{attribute 'GeneratedUsingTerminal: IODEVICETYPE_ETHERCATPROT'}
{attribute addProperty BoxType "IODEVICETYPE_ETHERCATPROT"}
{attribute addProperty Id "Term_26_EK1100Term_26_EK1100_99E5D94A13Box_29_EP1008_0001EP1008_78E8D3DD12Box_30_EP1008_0001EP1008_78E8D3DD12Box_31_EP1008_0001EP1008_78E8D3DD12Box_32_EP1008_0001EP1008_78E8D3DD12Box_33_EP1008_0001EP1008_78E8D3DD12Box_34_EP1008_0001EP1008_78E8D3DD12Box_35_EP1008_0001EP1008_78E8D3DD12Box_36_EP1008_0001EP1008_78E8D3DD12Box_37_EP1008_0001EP1008_78E8D3DD12Box_38_EP1008_0001EP1008_78E8D3DD12SyncUnitsSyncUnits_1397309536InputsInputs_A65FACA410OutputsOutputs_23C0ED1D6InfoDataInfoData_84133AC922"}
{attribute addProperty CRC "3568369493"}
{attribute addProperty Size "207"}
{attribute addProperty Name "Device 2 (EtherCAT)"}
TYPE Device_2_EtherCAT_D4B0FF55 EXTENDS TcoIo.EtcMasterBase_62654B43 :
STRUCT
	{attribute addProperty Name "Term 26 (EK1100)"}
	{attribute addProperty PreviousPort "Device 2 (EtherCAT) : Master"}
	Term_26_EK1100 : Term_26_EK1100_99E5D94A;
	{attribute addProperty Name "Box 29 (EP1008-0001)"}
	{attribute addProperty PreviousPort "Term 28 (EK1110) : B"}
	Box_29_EP1008_0001 : EP1008_78E8D3DD;
	{attribute addProperty Name "Box 30 (EP1008-0001)"}
	{attribute addProperty PreviousPort "Box 29 (EP1008-0001) : B"}
	Box_30_EP1008_0001 : EP1008_78E8D3DD;
	{attribute addProperty Name "Box 31 (EP1008-0001)"}
	{attribute addProperty PreviousPort "Box 30 (EP1008-0001) : B"}
	Box_31_EP1008_0001 : EP1008_78E8D3DD;
	{attribute addProperty Name "Box 32 (EP1008-0001)"}
	{attribute addProperty PreviousPort "Box 31 (EP1008-0001) : B"}
	Box_32_EP1008_0001 : EP1008_78E8D3DD;
	{attribute addProperty Name "Box 33 (EP1008-0001)"}
	{attribute addProperty PreviousPort "Box 32 (EP1008-0001) : B"}
	Box_33_EP1008_0001 : EP1008_78E8D3DD;
	{attribute addProperty Name "Box 34 (EP1008-0001)"}
	{attribute addProperty PreviousPort "Box 33 (EP1008-0001) : B"}
	Box_34_EP1008_0001 : EP1008_78E8D3DD;
	{attribute addProperty Name "Box 35 (EP1008-0001)"}
	{attribute addProperty PreviousPort "Box 34 (EP1008-0001) : B"}
	Box_35_EP1008_0001 : EP1008_78E8D3DD;
	{attribute addProperty Name "Box 36 (EP1008-0001)"}
	{attribute addProperty PreviousPort "Box 35 (EP1008-0001) : B"}
	Box_36_EP1008_0001 : EP1008_78E8D3DD;
	{attribute addProperty Name "Box 37 (EP1008-0001)"}
	{attribute addProperty PreviousPort "Box 36 (EP1008-0001) : B"}
	Box_37_EP1008_0001 : EP1008_78E8D3DD;
	{attribute addProperty Name "Box 38 (EP1008-0001)"}
	{attribute addProperty PreviousPort "Box 37 (EP1008-0001) : B"}
	Box_38_EP1008_0001 : EP1008_78E8D3DD;
	{attribute addProperty Name "SyncUnits"}
	SyncUnits : SyncUnits_13973095;
	{attribute addProperty Name "Inputs"}
	Inputs : TcoIo.Inputs_A65FACA4;
	{attribute addProperty Name "Outputs"}
	Outputs : TcoIo.Outputs_23C0ED1D;
	{attribute addProperty Name "InfoData"}
	InfoData : TcoIo.InfoData_84133AC9;
END_STRUCT
END_TYPE

(* stored: Version 1.2.0.0, ProductVersion 3.1.4024.11
   DUT Device_2_EtherCAT_D4B0FF55: Id {e4fa21fc-bc12-0c8a-139a-38541bd072b6} *)
